{attribute 'qualified_only'}
{attribute 'strict'}
{attribute 'to_string'}
TYPE enProductTypes :
(
	LK3G3_4G0C := 0,
	LK3G3_4L0A := 1
);
END_TYPE

(* stored: Version 1.1.0.1, ProductVersion 3.1.4024.10
   EnumerationTextList enProductTypes: Id {9264446b-380e-4d05-ba05-c3cb4b9e98c4} *)
